// TIA Portal V15.1 export
// export: Created 2024-06-21T08:41:23.5653437Z, ExportSetting WithDefaults, DisplayName Totally Integrated Automation Portal, DisplayVersion V15.1 Update 5, DisplayName TIA Portal Openness, DisplayVersion V15.1 Update 5, DisplayName SINAMICS Startdrive Advanced, DisplayVersion V15.1, DisplayName G130, G150, S120, S150, SINAMICS MV, S210, DisplayVersion V15.1, DisplayName G110M, G120, G120C, G120D, G120P, DisplayVersion V15.1, DisplayName STEP 7 Professional, DisplayVersion V15.1 Update 5, DisplayName STEP 7 Safety, DisplayVersion V15.1, DisplayName WinCC Professional, DisplayVersion V15.1 Update 5, DisplayName SIMATIC Visualization Architect, DisplayVersion V15.1
FUNCTION "209210ZS01AS" : Void   // FC322, FBD
TITLE = 209210ZS01AS Panels
{ S7_Optimized_Access := 'TRUE' }
AUTHOR : VCC
VERSION : 0.1
// stored: AutoNumber false, IsIECCheckEnabled false, SetENOAutomatically False, UDAEnableTagReadback false
   VAR_OUTPUT
      O_AlarmA : Bool;   // Alarm A
      O_AlarmB : Bool;   // Alarm B
      O_AlarmC : Bool;   // Alarm C
      O_AlarmD : Bool;   // Alarm D
      O_AlarmABCondition : Bool;   // Alarm AB condition
      H_IAnim : Word;   // For animation of icon
   END_VAR
BEGIN

REGION Network 1: **** --------------------- Pushbuttons Equipment 209210AS10 --------------------- ****
END_REGION

REGION Network 2: **** 4.3 - Machine status - Operator Selection **** Pushbutton 210CHB21 Holdback Down
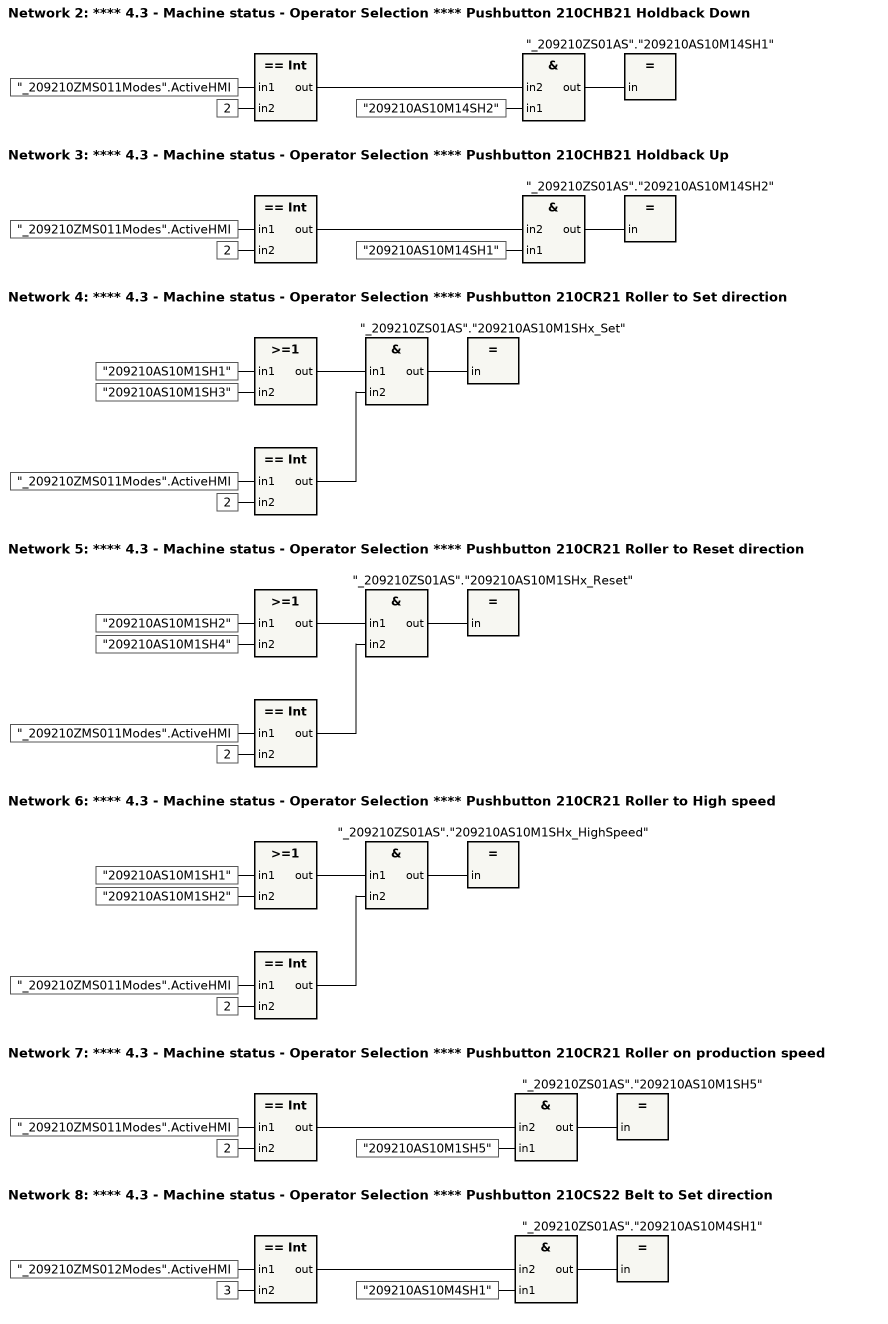
   "_209210ZS01AS"."209210AS10M14SH1" := ("_209210ZMS011Modes".ActiveHMI = 2) AND "209210AS10M14SH2";
END_REGION

REGION Network 3: **** 4.3 - Machine status - Operator Selection **** Pushbutton 210CHB21 Holdback Up
   "_209210ZS01AS"."209210AS10M14SH2" := ("_209210ZMS011Modes".ActiveHMI = 2) AND "209210AS10M14SH1";
END_REGION

REGION Network 4: **** 4.3 - Machine status - Operator Selection **** Pushbutton 210CR21 Roller to Set direction
   "_209210ZS01AS"."209210AS10M1SHx_Set" := ("209210AS10M1SH1" OR "209210AS10M1SH3") AND ("_209210ZMS011Modes".ActiveHMI = 2);
END_REGION

REGION Network 5: **** 4.3 - Machine status - Operator Selection **** Pushbutton 210CR21 Roller to Reset direction
   "_209210ZS01AS"."209210AS10M1SHx_Reset" := ("209210AS10M1SH2" OR "209210AS10M1SH4") AND ("_209210ZMS011Modes".ActiveHMI = 2);
END_REGION

REGION Network 6: **** 4.3 - Machine status - Operator Selection **** Pushbutton 210CR21 Roller to High speed
   "_209210ZS01AS"."209210AS10M1SHx_HighSpeed" := ("209210AS10M1SH1" OR "209210AS10M1SH2") AND ("_209210ZMS011Modes".ActiveHMI = 2);
END_REGION

REGION Network 7: **** 4.3 - Machine status - Operator Selection **** Pushbutton 210CR21 Roller on production speed
   "_209210ZS01AS"."209210AS10M1SH5" := ("_209210ZMS011Modes".ActiveHMI = 2) AND "209210AS10M1SH5";
END_REGION

REGION Network 8: **** 4.3 - Machine status - Operator Selection **** Pushbutton 210CS22 Belt to Set direction
   "_209210ZS01AS"."209210AS10M4SH1" := ("_209210ZMS012Modes".ActiveHMI = 3) AND "209210AS10M4SH1";
END_REGION

REGION Network 9: **** 4.3 - Machine status - Operator Selection **** Pushbutton 210CS22 Belt to Reset direction
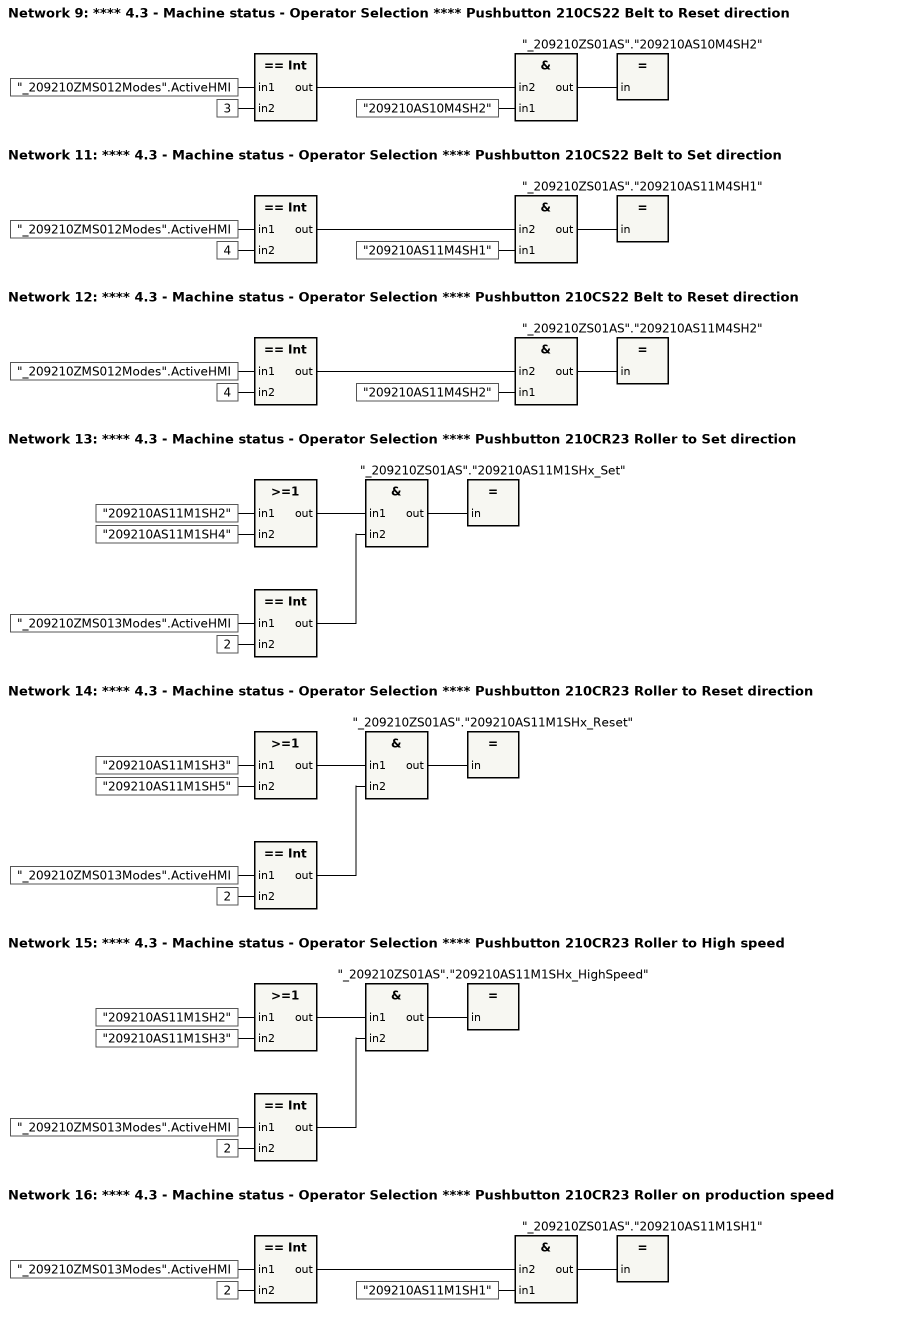
   "_209210ZS01AS"."209210AS10M4SH2" := ("_209210ZMS012Modes".ActiveHMI = 3) AND "209210AS10M4SH2";
END_REGION

REGION Network 10: **** --------------------- Pushbuttons Equipment 209210AS11 --------------------- ****
END_REGION

REGION Network 11: **** 4.3 - Machine status - Operator Selection **** Pushbutton 210CS22 Belt to Set direction
   "_209210ZS01AS"."209210AS11M4SH1" := ("_209210ZMS012Modes".ActiveHMI = 4) AND "209210AS11M4SH1";
END_REGION

REGION Network 12: **** 4.3 - Machine status - Operator Selection **** Pushbutton 210CS22 Belt to Reset direction
   "_209210ZS01AS"."209210AS11M4SH2" := ("_209210ZMS012Modes".ActiveHMI = 4) AND "209210AS11M4SH2";
END_REGION

REGION Network 13: **** 4.3 - Machine status - Operator Selection **** Pushbutton 210CR23 Roller to Set direction
   "_209210ZS01AS"."209210AS11M1SHx_Set" := ("209210AS11M1SH2" OR "209210AS11M1SH4") AND ("_209210ZMS013Modes".ActiveHMI = 2);
END_REGION

REGION Network 14: **** 4.3 - Machine status - Operator Selection **** Pushbutton 210CR23 Roller to Reset direction
   "_209210ZS01AS"."209210AS11M1SHx_Reset" := ("209210AS11M1SH3" OR "209210AS11M1SH5") AND ("_209210ZMS013Modes".ActiveHMI = 2);
END_REGION

REGION Network 15: **** 4.3 - Machine status - Operator Selection **** Pushbutton 210CR23 Roller to High speed
   "_209210ZS01AS"."209210AS11M1SHx_HighSpeed" := ("209210AS11M1SH2" OR "209210AS11M1SH3") AND ("_209210ZMS013Modes".ActiveHMI = 2);
END_REGION

REGION Network 16: **** 4.3 - Machine status - Operator Selection **** Pushbutton 210CR23 Roller on production speed
   "_209210ZS01AS"."209210AS11M1SH1" := ("_209210ZMS013Modes".ActiveHMI = 2) AND "209210AS11M1SH1";
END_REGION

REGION Network 17: **** -------------------------------------------------- ****
END_REGION

REGION Network 18: **** 4.6 - Machine status - Indications **** Icon animation
   // Icon animation
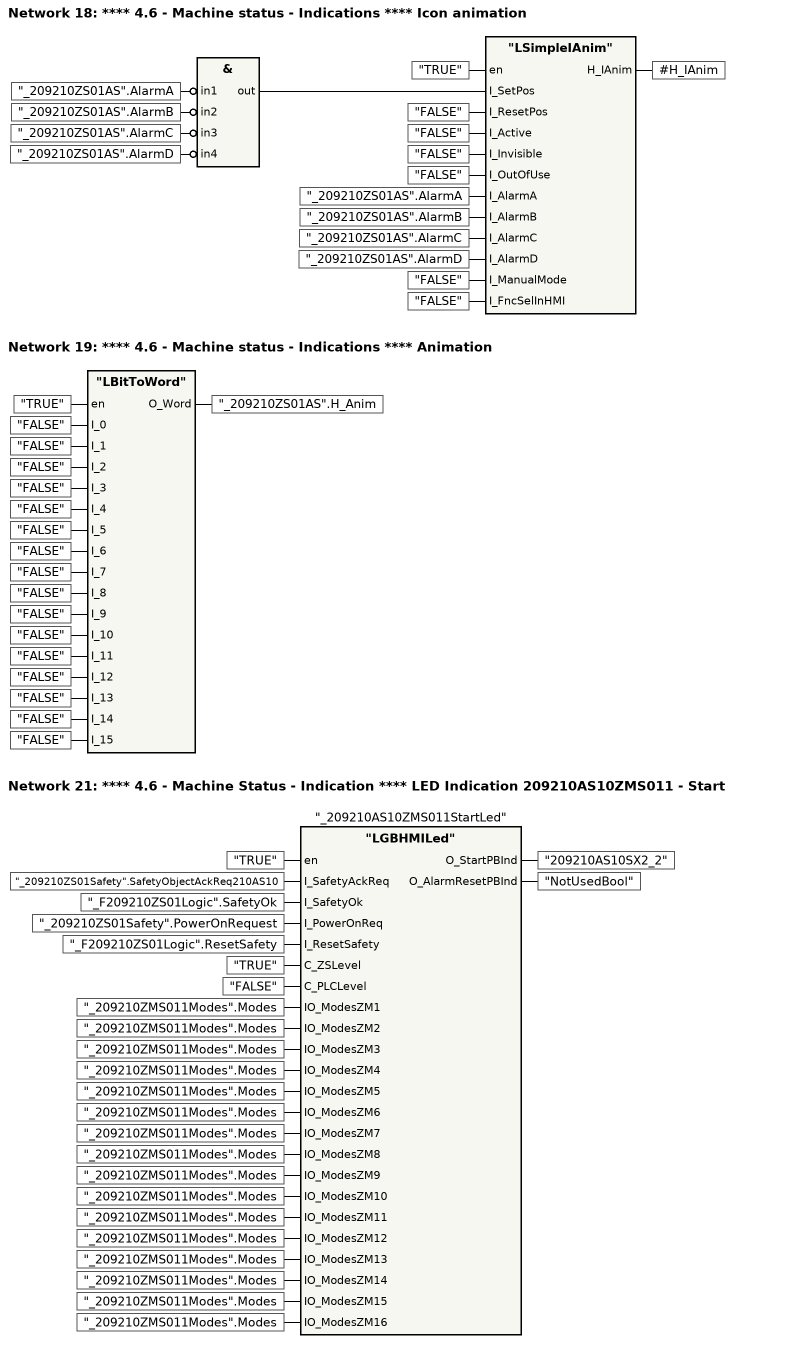
   IF "TRUE" THEN
       "LSimpleIAnim"(I_SetPos := NOT "_209210ZS01AS".AlarmA AND NOT "_209210ZS01AS".AlarmB AND NOT "_209210ZS01AS".AlarmC AND NOT "_209210ZS01AS".AlarmD,
                      I_ResetPos := "FALSE",
                      I_Active := "FALSE",
                      I_Invisible := "FALSE",
                      I_OutOfUse := "FALSE",
                      I_AlarmA := "_209210ZS01AS".AlarmA,
                      I_AlarmB := "_209210ZS01AS".AlarmB,
                      I_AlarmC := "_209210ZS01AS".AlarmC,
                      I_AlarmD := "_209210ZS01AS".AlarmD,
                      I_ManualMode := "FALSE",
                      I_FncSelInHMI := "FALSE",
                      H_IAnim => #H_IAnim);
   END_IF;
END_REGION

REGION Network 19: **** 4.6 - Machine status - Indications **** Animation
   // Animation
   IF "TRUE" THEN
       "LBitToWord"(I_0 := "FALSE",
                    I_1 := "FALSE",
                    I_2 := "FALSE",
                    I_3 := "FALSE",
                    I_4 := "FALSE",
                    I_5 := "FALSE",
                    I_6 := "FALSE",
                    I_7 := "FALSE",
                    I_8 := "FALSE",
                    I_9 := "FALSE",
                    I_10 := "FALSE",
                    I_11 := "FALSE",
                    I_12 := "FALSE",
                    I_13 := "FALSE",
                    I_14 := "FALSE",
                    I_15 := "FALSE",
                    O_Word => "_209210ZS01AS".H_Anim);
   END_IF;
END_REGION

NETWORK
TITLE = **** 4.6 - Machine Status - Indications **** Animation DB number
// DB number
      OPN   "_209210ZS01AS";
      L     DBNO;
      T     "_209210ZS01AS".H_DBnr;

REGION Network 21: **** 4.6 - Machine Status - Indication **** LED Indication 209210AS10ZMS011 - Start
   // The Module handles indications for Start and Reset buttons
   IF "TRUE" THEN
       "_209210AS10ZMS011StartLed"(I_SafetyAckReq := "_209210ZS01Safety".SafetyObjectAckReq210AS10,   // "LGBHMILed"
                               I_SafetyOk := "_F209210ZS01Logic".SafetyOk,
                               I_PowerOnReq := "_209210ZS01Safety".PowerOnRequest,
                               I_ResetSafety := "_F209210ZS01Logic".ResetSafety,
                               C_ZSLevel := "TRUE",
                               C_PLCLevel := "FALSE",
                               IO_ModesZM1 := "_209210ZMS011Modes".Modes,
                               IO_ModesZM2 := "_209210ZMS011Modes".Modes,
                               IO_ModesZM3 := "_209210ZMS011Modes".Modes,
                               IO_ModesZM4 := "_209210ZMS011Modes".Modes,
                               IO_ModesZM5 := "_209210ZMS011Modes".Modes,
                               IO_ModesZM6 := "_209210ZMS011Modes".Modes,
                               IO_ModesZM7 := "_209210ZMS011Modes".Modes,
                               IO_ModesZM8 := "_209210ZMS011Modes".Modes,
                               IO_ModesZM9 := "_209210ZMS011Modes".Modes,
                               IO_ModesZM10 := "_209210ZMS011Modes".Modes,
                               IO_ModesZM11 := "_209210ZMS011Modes".Modes,
                               IO_ModesZM12 := "_209210ZMS011Modes".Modes,
                               IO_ModesZM13 := "_209210ZMS011Modes".Modes,
                               IO_ModesZM14 := "_209210ZMS011Modes".Modes,
                               IO_ModesZM15 := "_209210ZMS011Modes".Modes,
                               IO_ModesZM16 := "_209210ZMS011Modes".Modes,
                               O_StartPBInd => "209210AS10SX2_2",
                               O_AlarmResetPBInd => "NotUsedBool");
   END_IF;
END_REGION

REGION Network 22: **** 4.6 - Machine Status - Indication **** LED Indication 209210AS10ZMS012 - Start
   // The Module handles indications for Start and Reset buttons
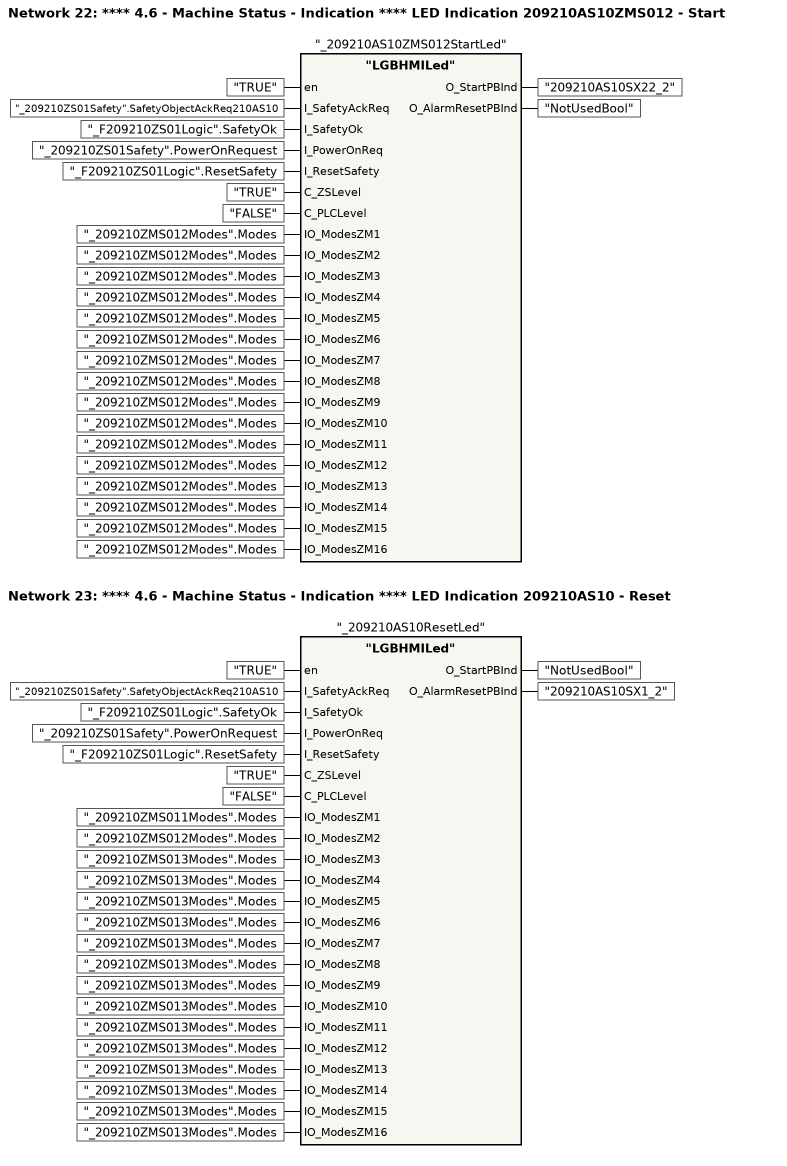
   IF "TRUE" THEN
       "_209210AS10ZMS012StartLed"(I_SafetyAckReq := "_209210ZS01Safety".SafetyObjectAckReq210AS10,   // "LGBHMILed"
                               I_SafetyOk := "_F209210ZS01Logic".SafetyOk,
                               I_PowerOnReq := "_209210ZS01Safety".PowerOnRequest,
                               I_ResetSafety := "_F209210ZS01Logic".ResetSafety,
                               C_ZSLevel := "TRUE",
                               C_PLCLevel := "FALSE",
                               IO_ModesZM1 := "_209210ZMS012Modes".Modes,
                               IO_ModesZM2 := "_209210ZMS012Modes".Modes,
                               IO_ModesZM3 := "_209210ZMS012Modes".Modes,
                               IO_ModesZM4 := "_209210ZMS012Modes".Modes,
                               IO_ModesZM5 := "_209210ZMS012Modes".Modes,
                               IO_ModesZM6 := "_209210ZMS012Modes".Modes,
                               IO_ModesZM7 := "_209210ZMS012Modes".Modes,
                               IO_ModesZM8 := "_209210ZMS012Modes".Modes,
                               IO_ModesZM9 := "_209210ZMS012Modes".Modes,
                               IO_ModesZM10 := "_209210ZMS012Modes".Modes,
                               IO_ModesZM11 := "_209210ZMS012Modes".Modes,
                               IO_ModesZM12 := "_209210ZMS012Modes".Modes,
                               IO_ModesZM13 := "_209210ZMS012Modes".Modes,
                               IO_ModesZM14 := "_209210ZMS012Modes".Modes,
                               IO_ModesZM15 := "_209210ZMS012Modes".Modes,
                               IO_ModesZM16 := "_209210ZMS012Modes".Modes,
                               O_StartPBInd => "209210AS10SX22_2",
                               O_AlarmResetPBInd => "NotUsedBool");
   END_IF;
END_REGION

REGION Network 23: **** 4.6 - Machine Status - Indication **** LED Indication 209210AS10 - Reset
   // The Module handles indications for Start and Reset buttons
   IF "TRUE" THEN
       "_209210AS10ResetLed"(I_SafetyAckReq := "_209210ZS01Safety".SafetyObjectAckReq210AS10,   // "LGBHMILed"
                             I_SafetyOk := "_F209210ZS01Logic".SafetyOk,
                             I_PowerOnReq := "_209210ZS01Safety".PowerOnRequest,
                             I_ResetSafety := "_F209210ZS01Logic".ResetSafety,
                             C_ZSLevel := "TRUE",
                             C_PLCLevel := "FALSE",
                             IO_ModesZM1 := "_209210ZMS011Modes".Modes,
                             IO_ModesZM2 := "_209210ZMS012Modes".Modes,
                             IO_ModesZM3 := "_209210ZMS013Modes".Modes,
                             IO_ModesZM4 := "_209210ZMS013Modes".Modes,
                             IO_ModesZM5 := "_209210ZMS013Modes".Modes,
                             IO_ModesZM6 := "_209210ZMS013Modes".Modes,
                             IO_ModesZM7 := "_209210ZMS013Modes".Modes,
                             IO_ModesZM8 := "_209210ZMS013Modes".Modes,
                             IO_ModesZM9 := "_209210ZMS013Modes".Modes,
                             IO_ModesZM10 := "_209210ZMS013Modes".Modes,
                             IO_ModesZM11 := "_209210ZMS013Modes".Modes,
                             IO_ModesZM12 := "_209210ZMS013Modes".Modes,
                             IO_ModesZM13 := "_209210ZMS013Modes".Modes,
                             IO_ModesZM14 := "_209210ZMS013Modes".Modes,
                             IO_ModesZM15 := "_209210ZMS013Modes".Modes,
                             IO_ModesZM16 := "_209210ZMS013Modes".Modes,
                             O_StartPBInd => "NotUsedBool",
                             O_AlarmResetPBInd => "209210AS10SX1_2");
   END_IF;
END_REGION

REGION Network 24: **** 4.6 - Machine Status - Indication **** LED Indication 209210AS11ZMS012 - Start
   // The Module handles indications for Start and Reset buttons
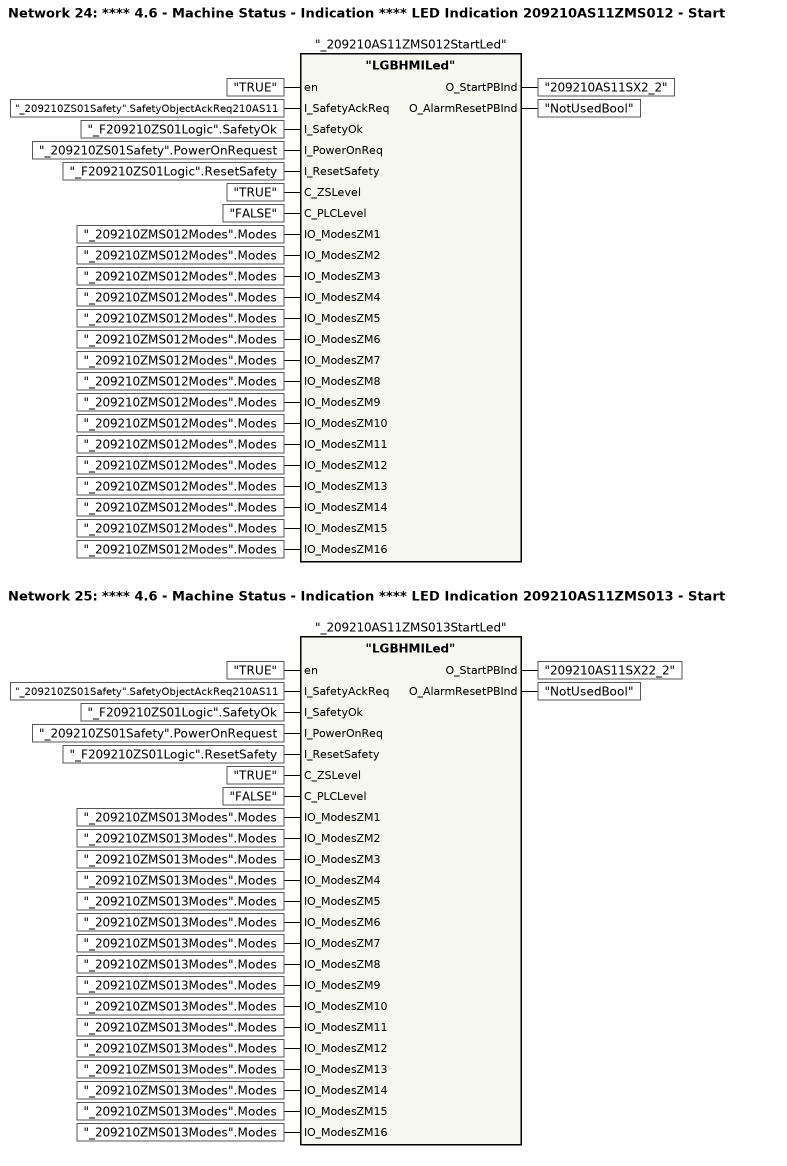
   IF "TRUE" THEN
       "_209210AS11ZMS012StartLed"(I_SafetyAckReq := "_209210ZS01Safety".SafetyObjectAckReq210AS11,   // "LGBHMILed"
                               I_SafetyOk := "_F209210ZS01Logic".SafetyOk,
                               I_PowerOnReq := "_209210ZS01Safety".PowerOnRequest,
                               I_ResetSafety := "_F209210ZS01Logic".ResetSafety,
                               C_ZSLevel := "TRUE",
                               C_PLCLevel := "FALSE",
                               IO_ModesZM1 := "_209210ZMS012Modes".Modes,
                               IO_ModesZM2 := "_209210ZMS012Modes".Modes,
                               IO_ModesZM3 := "_209210ZMS012Modes".Modes,
                               IO_ModesZM4 := "_209210ZMS012Modes".Modes,
                               IO_ModesZM5 := "_209210ZMS012Modes".Modes,
                               IO_ModesZM6 := "_209210ZMS012Modes".Modes,
                               IO_ModesZM7 := "_209210ZMS012Modes".Modes,
                               IO_ModesZM8 := "_209210ZMS012Modes".Modes,
                               IO_ModesZM9 := "_209210ZMS012Modes".Modes,
                               IO_ModesZM10 := "_209210ZMS012Modes".Modes,
                               IO_ModesZM11 := "_209210ZMS012Modes".Modes,
                               IO_ModesZM12 := "_209210ZMS012Modes".Modes,
                               IO_ModesZM13 := "_209210ZMS012Modes".Modes,
                               IO_ModesZM14 := "_209210ZMS012Modes".Modes,
                               IO_ModesZM15 := "_209210ZMS012Modes".Modes,
                               IO_ModesZM16 := "_209210ZMS012Modes".Modes,
                               O_StartPBInd => "209210AS11SX2_2",
                               O_AlarmResetPBInd => "NotUsedBool");
   END_IF;
END_REGION

REGION Network 25: **** 4.6 - Machine Status - Indication **** LED Indication 209210AS11ZMS013 - Start
   // The Module handles indications for Start and Reset buttons
   IF "TRUE" THEN
       "_209210AS11ZMS013StartLed"(I_SafetyAckReq := "_209210ZS01Safety".SafetyObjectAckReq210AS11,   // "LGBHMILed"
                               I_SafetyOk := "_F209210ZS01Logic".SafetyOk,
                               I_PowerOnReq := "_209210ZS01Safety".PowerOnRequest,
                               I_ResetSafety := "_F209210ZS01Logic".ResetSafety,
                               C_ZSLevel := "TRUE",
                               C_PLCLevel := "FALSE",
                               IO_ModesZM1 := "_209210ZMS013Modes".Modes,
                               IO_ModesZM2 := "_209210ZMS013Modes".Modes,
                               IO_ModesZM3 := "_209210ZMS013Modes".Modes,
                               IO_ModesZM4 := "_209210ZMS013Modes".Modes,
                               IO_ModesZM5 := "_209210ZMS013Modes".Modes,
                               IO_ModesZM6 := "_209210ZMS013Modes".Modes,
                               IO_ModesZM7 := "_209210ZMS013Modes".Modes,
                               IO_ModesZM8 := "_209210ZMS013Modes".Modes,
                               IO_ModesZM9 := "_209210ZMS013Modes".Modes,
                               IO_ModesZM10 := "_209210ZMS013Modes".Modes,
                               IO_ModesZM11 := "_209210ZMS013Modes".Modes,
                               IO_ModesZM12 := "_209210ZMS013Modes".Modes,
                               IO_ModesZM13 := "_209210ZMS013Modes".Modes,
                               IO_ModesZM14 := "_209210ZMS013Modes".Modes,
                               IO_ModesZM15 := "_209210ZMS013Modes".Modes,
                               IO_ModesZM16 := "_209210ZMS013Modes".Modes,
                               O_StartPBInd => "209210AS11SX22_2",
                               O_AlarmResetPBInd => "NotUsedBool");
   END_IF;
END_REGION

REGION Network 26: **** 4.6 - Machine Status - Indication **** LED Indication 209210AS11 - Reset
   // The Module handles indications for Start and Reset buttons
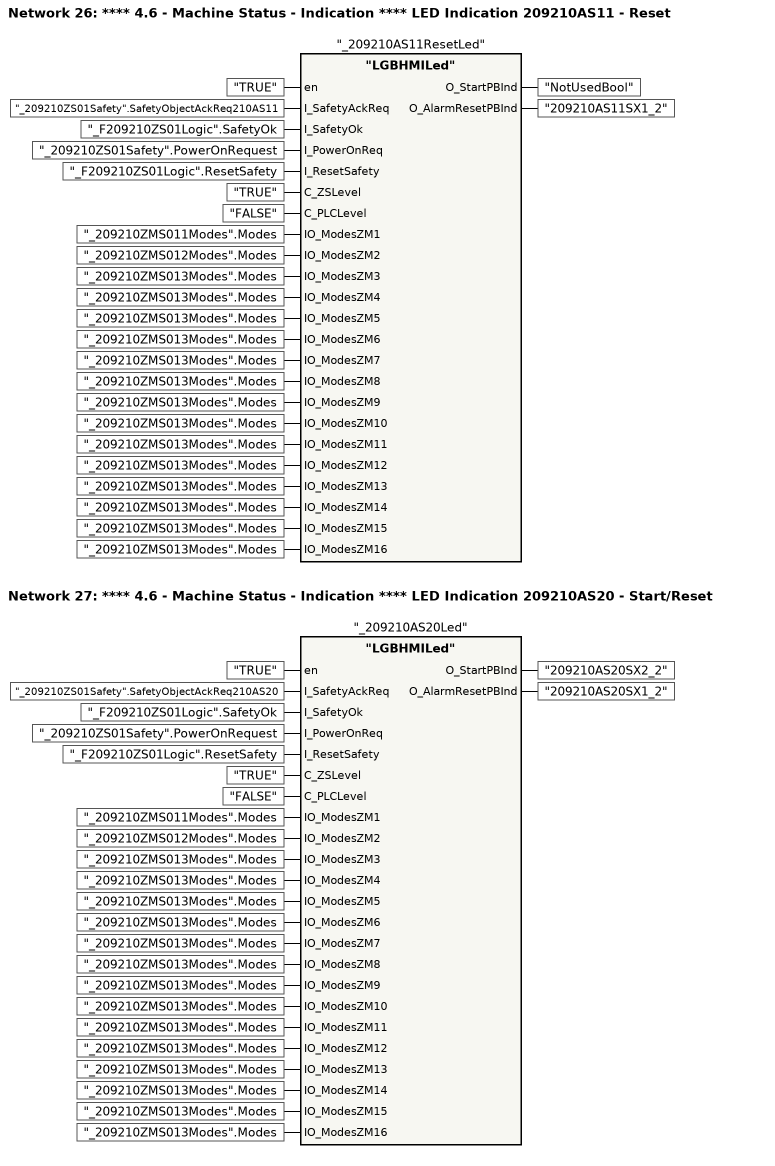
   IF "TRUE" THEN
       "_209210AS11ResetLed"(I_SafetyAckReq := "_209210ZS01Safety".SafetyObjectAckReq210AS11,   // "LGBHMILed"
                             I_SafetyOk := "_F209210ZS01Logic".SafetyOk,
                             I_PowerOnReq := "_209210ZS01Safety".PowerOnRequest,
                             I_ResetSafety := "_F209210ZS01Logic".ResetSafety,
                             C_ZSLevel := "TRUE",
                             C_PLCLevel := "FALSE",
                             IO_ModesZM1 := "_209210ZMS011Modes".Modes,
                             IO_ModesZM2 := "_209210ZMS012Modes".Modes,
                             IO_ModesZM3 := "_209210ZMS013Modes".Modes,
                             IO_ModesZM4 := "_209210ZMS013Modes".Modes,
                             IO_ModesZM5 := "_209210ZMS013Modes".Modes,
                             IO_ModesZM6 := "_209210ZMS013Modes".Modes,
                             IO_ModesZM7 := "_209210ZMS013Modes".Modes,
                             IO_ModesZM8 := "_209210ZMS013Modes".Modes,
                             IO_ModesZM9 := "_209210ZMS013Modes".Modes,
                             IO_ModesZM10 := "_209210ZMS013Modes".Modes,
                             IO_ModesZM11 := "_209210ZMS013Modes".Modes,
                             IO_ModesZM12 := "_209210ZMS013Modes".Modes,
                             IO_ModesZM13 := "_209210ZMS013Modes".Modes,
                             IO_ModesZM14 := "_209210ZMS013Modes".Modes,
                             IO_ModesZM15 := "_209210ZMS013Modes".Modes,
                             IO_ModesZM16 := "_209210ZMS013Modes".Modes,
                             O_StartPBInd => "NotUsedBool",
                             O_AlarmResetPBInd => "209210AS11SX1_2");
   END_IF;
END_REGION

REGION Network 27: **** 4.6 - Machine Status - Indication **** LED Indication 209210AS20 - Start/Reset
   // The Module handles indications for Start and Reset buttons
   IF "TRUE" THEN
       "_209210AS20Led"(I_SafetyAckReq := "_209210ZS01Safety".SafetyObjectAckReq210AS20,   // "LGBHMILed"
                        I_SafetyOk := "_F209210ZS01Logic".SafetyOk,
                        I_PowerOnReq := "_209210ZS01Safety".PowerOnRequest,
                        I_ResetSafety := "_F209210ZS01Logic".ResetSafety,
                        C_ZSLevel := "TRUE",
                        C_PLCLevel := "FALSE",
                        IO_ModesZM1 := "_209210ZMS011Modes".Modes,
                        IO_ModesZM2 := "_209210ZMS012Modes".Modes,
                        IO_ModesZM3 := "_209210ZMS013Modes".Modes,
                        IO_ModesZM4 := "_209210ZMS013Modes".Modes,
                        IO_ModesZM5 := "_209210ZMS013Modes".Modes,
                        IO_ModesZM6 := "_209210ZMS013Modes".Modes,
                        IO_ModesZM7 := "_209210ZMS013Modes".Modes,
                        IO_ModesZM8 := "_209210ZMS013Modes".Modes,
                        IO_ModesZM9 := "_209210ZMS013Modes".Modes,
                        IO_ModesZM10 := "_209210ZMS013Modes".Modes,
                        IO_ModesZM11 := "_209210ZMS013Modes".Modes,
                        IO_ModesZM12 := "_209210ZMS013Modes".Modes,
                        IO_ModesZM13 := "_209210ZMS013Modes".Modes,
                        IO_ModesZM14 := "_209210ZMS013Modes".Modes,
                        IO_ModesZM15 := "_209210ZMS013Modes".Modes,
                        IO_ModesZM16 := "_209210ZMS013Modes".Modes,
                        O_StartPBInd => "209210AS20SX2_2",
                        O_AlarmResetPBInd => "209210AS20SX1_2");
   END_IF;
END_REGION

REGION Network 28: **** 4.6 - Machine Status - Indication **** LED Indication 209210AS40 - Start/Reset
   // The Module handles indications for Start and Reset buttons
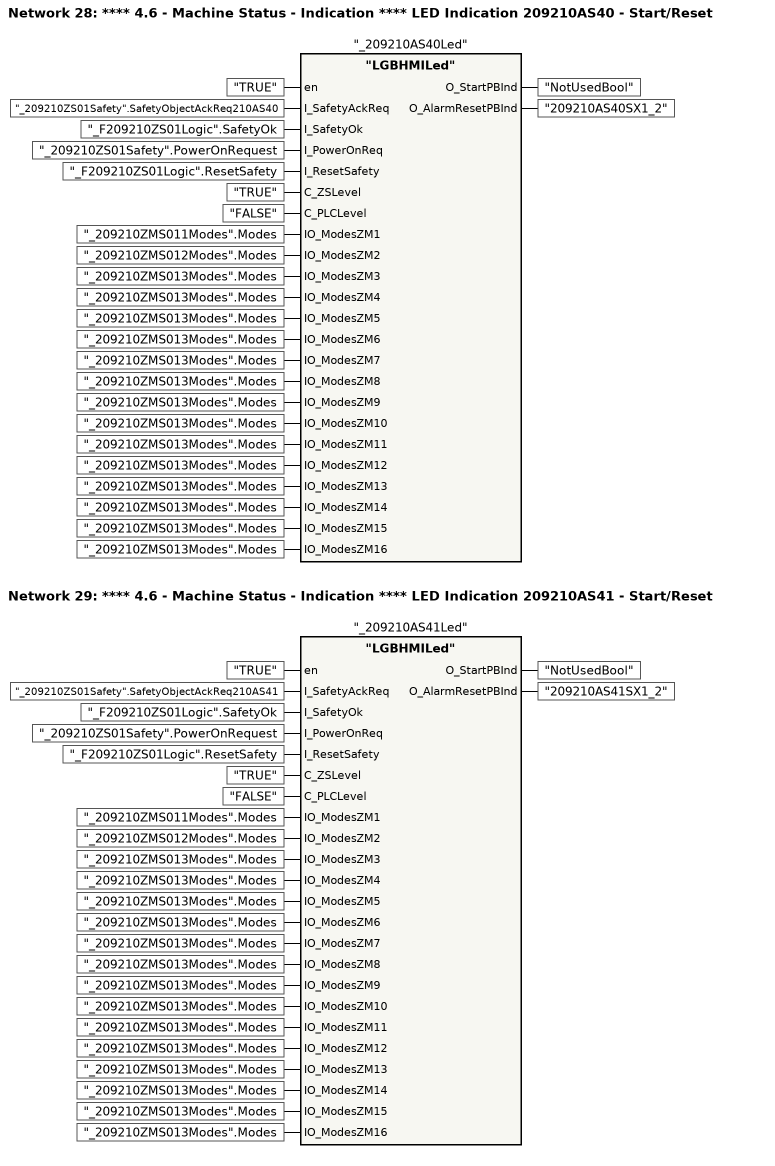
   IF "TRUE" THEN
       "_209210AS40Led"(I_SafetyAckReq := "_209210ZS01Safety".SafetyObjectAckReq210AS40,   // "LGBHMILed"
                        I_SafetyOk := "_F209210ZS01Logic".SafetyOk,
                        I_PowerOnReq := "_209210ZS01Safety".PowerOnRequest,
                        I_ResetSafety := "_F209210ZS01Logic".ResetSafety,
                        C_ZSLevel := "TRUE",
                        C_PLCLevel := "FALSE",
                        IO_ModesZM1 := "_209210ZMS011Modes".Modes,
                        IO_ModesZM2 := "_209210ZMS012Modes".Modes,
                        IO_ModesZM3 := "_209210ZMS013Modes".Modes,
                        IO_ModesZM4 := "_209210ZMS013Modes".Modes,
                        IO_ModesZM5 := "_209210ZMS013Modes".Modes,
                        IO_ModesZM6 := "_209210ZMS013Modes".Modes,
                        IO_ModesZM7 := "_209210ZMS013Modes".Modes,
                        IO_ModesZM8 := "_209210ZMS013Modes".Modes,
                        IO_ModesZM9 := "_209210ZMS013Modes".Modes,
                        IO_ModesZM10 := "_209210ZMS013Modes".Modes,
                        IO_ModesZM11 := "_209210ZMS013Modes".Modes,
                        IO_ModesZM12 := "_209210ZMS013Modes".Modes,
                        IO_ModesZM13 := "_209210ZMS013Modes".Modes,
                        IO_ModesZM14 := "_209210ZMS013Modes".Modes,
                        IO_ModesZM15 := "_209210ZMS013Modes".Modes,
                        IO_ModesZM16 := "_209210ZMS013Modes".Modes,
                        O_StartPBInd => "NotUsedBool",
                        O_AlarmResetPBInd => "209210AS40SX1_2");
   END_IF;
END_REGION

REGION Network 29: **** 4.6 - Machine Status - Indication **** LED Indication 209210AS41 - Start/Reset
   // The Module handles indications for Start and Reset buttons
   IF "TRUE" THEN
       "_209210AS41Led"(I_SafetyAckReq := "_209210ZS01Safety".SafetyObjectAckReq210AS41,   // "LGBHMILed"
                        I_SafetyOk := "_F209210ZS01Logic".SafetyOk,
                        I_PowerOnReq := "_209210ZS01Safety".PowerOnRequest,
                        I_ResetSafety := "_F209210ZS01Logic".ResetSafety,
                        C_ZSLevel := "TRUE",
                        C_PLCLevel := "FALSE",
                        IO_ModesZM1 := "_209210ZMS011Modes".Modes,
                        IO_ModesZM2 := "_209210ZMS012Modes".Modes,
                        IO_ModesZM3 := "_209210ZMS013Modes".Modes,
                        IO_ModesZM4 := "_209210ZMS013Modes".Modes,
                        IO_ModesZM5 := "_209210ZMS013Modes".Modes,
                        IO_ModesZM6 := "_209210ZMS013Modes".Modes,
                        IO_ModesZM7 := "_209210ZMS013Modes".Modes,
                        IO_ModesZM8 := "_209210ZMS013Modes".Modes,
                        IO_ModesZM9 := "_209210ZMS013Modes".Modes,
                        IO_ModesZM10 := "_209210ZMS013Modes".Modes,
                        IO_ModesZM11 := "_209210ZMS013Modes".Modes,
                        IO_ModesZM12 := "_209210ZMS013Modes".Modes,
                        IO_ModesZM13 := "_209210ZMS013Modes".Modes,
                        IO_ModesZM14 := "_209210ZMS013Modes".Modes,
                        IO_ModesZM15 := "_209210ZMS013Modes".Modes,
                        IO_ModesZM16 := "_209210ZMS013Modes".Modes,
                        O_StartPBInd => "NotUsedBool",
                        O_AlarmResetPBInd => "209210AS41SX1_2");
   END_IF;
END_REGION

REGION Network 30: **** 4.6 - Machine Status - Indication **** LED Indication 209210ASH01 - Start/Reset
   // The Module handles indications for Start and Reset buttons
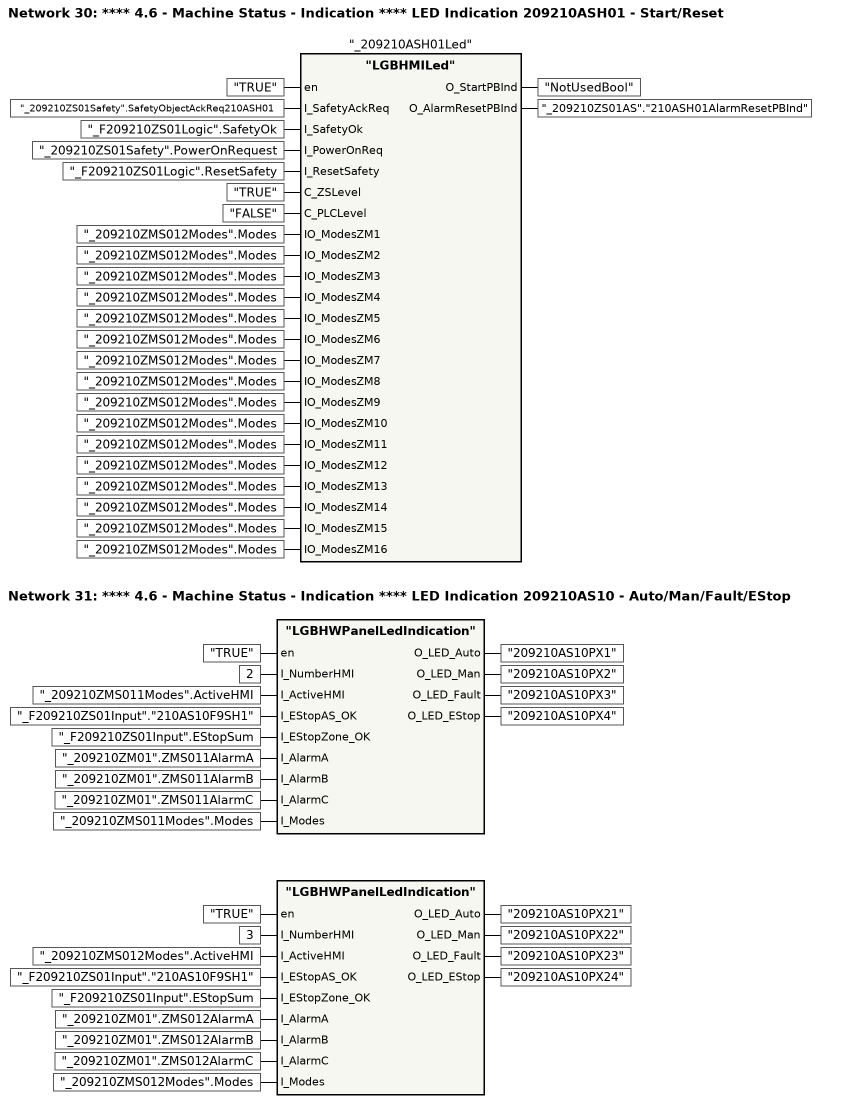
   IF "TRUE" THEN
       "_209210ASH01Led"(I_SafetyAckReq := "_209210ZS01Safety".SafetyObjectAckReq210ASH01,   // "LGBHMILed"
                         I_SafetyOk := "_F209210ZS01Logic".SafetyOk,
                         I_PowerOnReq := "_209210ZS01Safety".PowerOnRequest,
                         I_ResetSafety := "_F209210ZS01Logic".ResetSafety,
                         C_ZSLevel := "TRUE",
                         C_PLCLevel := "FALSE",
                         IO_ModesZM1 := "_209210ZMS012Modes".Modes,
                         IO_ModesZM2 := "_209210ZMS012Modes".Modes,
                         IO_ModesZM3 := "_209210ZMS012Modes".Modes,
                         IO_ModesZM4 := "_209210ZMS012Modes".Modes,
                         IO_ModesZM5 := "_209210ZMS012Modes".Modes,
                         IO_ModesZM6 := "_209210ZMS012Modes".Modes,
                         IO_ModesZM7 := "_209210ZMS012Modes".Modes,
                         IO_ModesZM8 := "_209210ZMS012Modes".Modes,
                         IO_ModesZM9 := "_209210ZMS012Modes".Modes,
                         IO_ModesZM10 := "_209210ZMS012Modes".Modes,
                         IO_ModesZM11 := "_209210ZMS012Modes".Modes,
                         IO_ModesZM12 := "_209210ZMS012Modes".Modes,
                         IO_ModesZM13 := "_209210ZMS012Modes".Modes,
                         IO_ModesZM14 := "_209210ZMS012Modes".Modes,
                         IO_ModesZM15 := "_209210ZMS012Modes".Modes,
                         IO_ModesZM16 := "_209210ZMS012Modes".Modes,
                         O_StartPBInd => "NotUsedBool",
                         O_AlarmResetPBInd => "_209210ZS01AS"."210ASH01AlarmResetPBInd");
   END_IF;
END_REGION

REGION Network 31: **** 4.6 - Machine Status - Indication **** LED Indication 209210AS10 - Auto/Man/Fault/EStop
   IF "TRUE" THEN
       "LGBHWPanelLedIndication"(I_NumberHMI := 2,
                               I_ActiveHMI := "_209210ZMS011Modes".ActiveHMI,
                               I_EStopAS_OK := "_F209210ZS01Input"."210AS10F9SH1",
                               I_EStopZone_OK := "_F209210ZS01Input".EStopSum,
                               I_AlarmA := "_209210ZM01".ZMS011AlarmA,
                               I_AlarmB := "_209210ZM01".ZMS011AlarmB,
                               I_AlarmC := "_209210ZM01".ZMS011AlarmC,
                               I_Modes := "_209210ZMS011Modes".Modes,
                               O_LED_Auto => "209210AS10PX1",
                               O_LED_Man => "209210AS10PX2",
                               O_LED_Fault => "209210AS10PX3",
                               O_LED_EStop => "209210AS10PX4");
   END_IF;
   IF "TRUE" THEN
       "LGBHWPanelLedIndication"(I_NumberHMI := 3,
                               I_ActiveHMI := "_209210ZMS012Modes".ActiveHMI,
                               I_EStopAS_OK := "_F209210ZS01Input"."210AS10F9SH1",
                               I_EStopZone_OK := "_F209210ZS01Input".EStopSum,
                               I_AlarmA := "_209210ZM01".ZMS012AlarmA,
                               I_AlarmB := "_209210ZM01".ZMS012AlarmB,
                               I_AlarmC := "_209210ZM01".ZMS012AlarmC,
                               I_Modes := "_209210ZMS012Modes".Modes,
                               O_LED_Auto => "209210AS10PX21",
                               O_LED_Man => "209210AS10PX22",
                               O_LED_Fault => "209210AS10PX23",
                               O_LED_EStop => "209210AS10PX24");
   END_IF;
END_REGION

REGION Network 32: **** 4.6 - Machine Status - Indication **** LED Indication 209210AS11 - Auto/Man/Fault/EStop
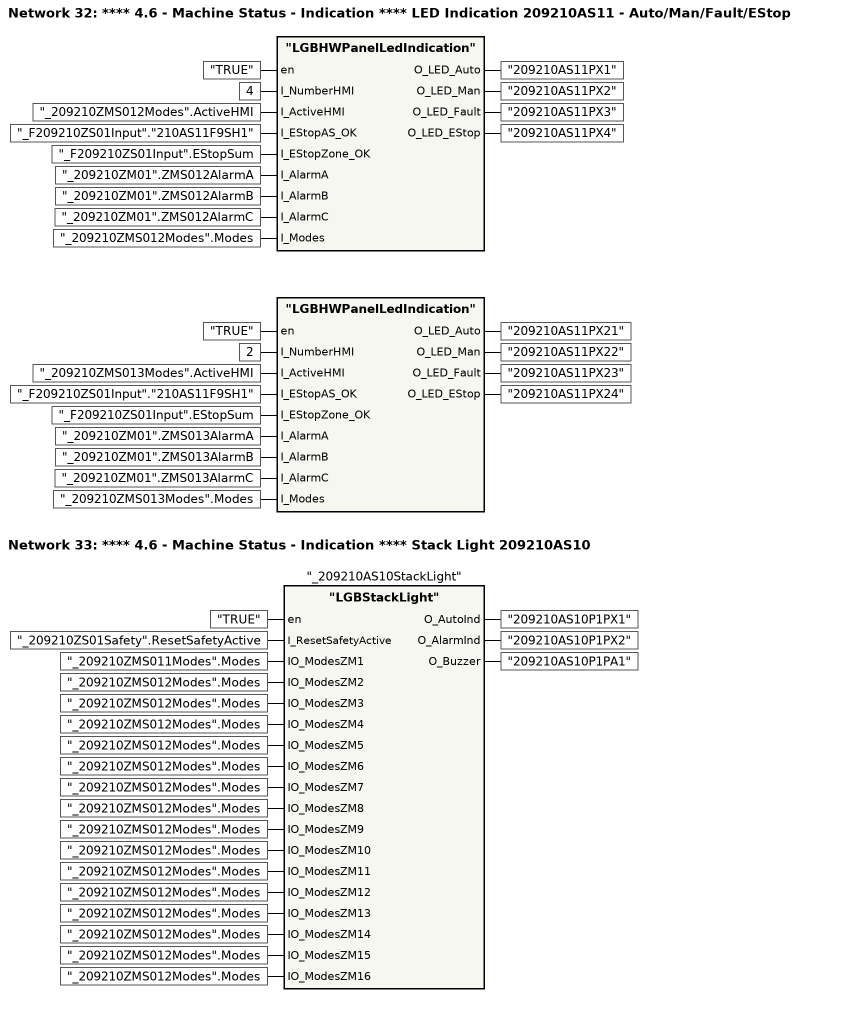
   IF "TRUE" THEN
       "LGBHWPanelLedIndication"(I_NumberHMI := 4,
                               I_ActiveHMI := "_209210ZMS012Modes".ActiveHMI,
                               I_EStopAS_OK := "_F209210ZS01Input"."210AS11F9SH1",
                               I_EStopZone_OK := "_F209210ZS01Input".EStopSum,
                               I_AlarmA := "_209210ZM01".ZMS012AlarmA,
                               I_AlarmB := "_209210ZM01".ZMS012AlarmB,
                               I_AlarmC := "_209210ZM01".ZMS012AlarmC,
                               I_Modes := "_209210ZMS012Modes".Modes,
                               O_LED_Auto => "209210AS11PX1",
                               O_LED_Man => "209210AS11PX2",
                               O_LED_Fault => "209210AS11PX3",
                               O_LED_EStop => "209210AS11PX4");
   END_IF;
   IF "TRUE" THEN
       "LGBHWPanelLedIndication"(I_NumberHMI := 2,
                               I_ActiveHMI := "_209210ZMS013Modes".ActiveHMI,
                               I_EStopAS_OK := "_F209210ZS01Input"."210AS11F9SH1",
                               I_EStopZone_OK := "_F209210ZS01Input".EStopSum,
                               I_AlarmA := "_209210ZM01".ZMS013AlarmA,
                               I_AlarmB := "_209210ZM01".ZMS013AlarmB,
                               I_AlarmC := "_209210ZM01".ZMS013AlarmC,
                               I_Modes := "_209210ZMS013Modes".Modes,
                               O_LED_Auto => "209210AS11PX21",
                               O_LED_Man => "209210AS11PX22",
                               O_LED_Fault => "209210AS11PX23",
                               O_LED_EStop => "209210AS11PX24");
   END_IF;
END_REGION

REGION Network 33: **** 4.6 - Machine Status - Indication **** Stack Light 209210AS10
   IF "TRUE" THEN
       "_209210AS10StackLight"(I_ResetSafetyActive := "_209210ZS01Safety".ResetSafetyActive,   // "LGBStackLight"
                               IO_ModesZM1 := "_209210ZMS011Modes".Modes,
                               IO_ModesZM2 := "_209210ZMS012Modes".Modes,
                               IO_ModesZM3 := "_209210ZMS012Modes".Modes,
                               IO_ModesZM4 := "_209210ZMS012Modes".Modes,
                               IO_ModesZM5 := "_209210ZMS012Modes".Modes,
                               IO_ModesZM6 := "_209210ZMS012Modes".Modes,
                               IO_ModesZM7 := "_209210ZMS012Modes".Modes,
                               IO_ModesZM8 := "_209210ZMS012Modes".Modes,
                               IO_ModesZM9 := "_209210ZMS012Modes".Modes,
                               IO_ModesZM10 := "_209210ZMS012Modes".Modes,
                               IO_ModesZM11 := "_209210ZMS012Modes".Modes,
                               IO_ModesZM12 := "_209210ZMS012Modes".Modes,
                               IO_ModesZM13 := "_209210ZMS012Modes".Modes,
                               IO_ModesZM14 := "_209210ZMS012Modes".Modes,
                               IO_ModesZM15 := "_209210ZMS012Modes".Modes,
                               IO_ModesZM16 := "_209210ZMS012Modes".Modes,
                               O_AutoInd => "209210AS10P1PX1",
                               O_AlarmInd => "209210AS10P1PX2",
                               O_Buzzer => "209210AS10P1PA1");
   END_IF;
END_REGION

REGION Network 34: **** 4.6 - Machine Status - Indication **** Stack Light 209210AS11
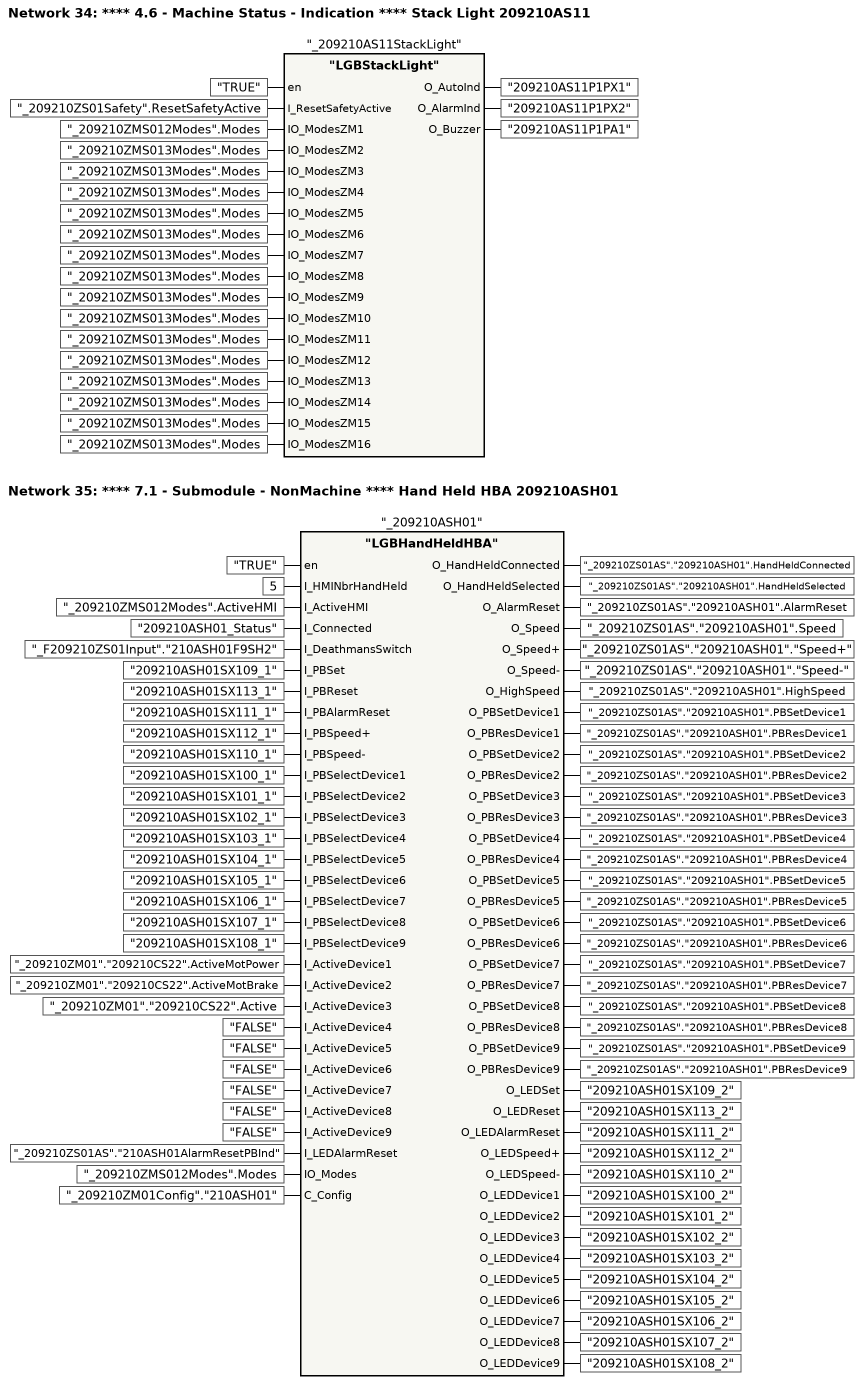
   IF "TRUE" THEN
       "_209210AS11StackLight"(I_ResetSafetyActive := "_209210ZS01Safety".ResetSafetyActive,   // "LGBStackLight"
                               IO_ModesZM1 := "_209210ZMS012Modes".Modes,
                               IO_ModesZM2 := "_209210ZMS013Modes".Modes,
                               IO_ModesZM3 := "_209210ZMS013Modes".Modes,
                               IO_ModesZM4 := "_209210ZMS013Modes".Modes,
                               IO_ModesZM5 := "_209210ZMS013Modes".Modes,
                               IO_ModesZM6 := "_209210ZMS013Modes".Modes,
                               IO_ModesZM7 := "_209210ZMS013Modes".Modes,
                               IO_ModesZM8 := "_209210ZMS013Modes".Modes,
                               IO_ModesZM9 := "_209210ZMS013Modes".Modes,
                               IO_ModesZM10 := "_209210ZMS013Modes".Modes,
                               IO_ModesZM11 := "_209210ZMS013Modes".Modes,
                               IO_ModesZM12 := "_209210ZMS013Modes".Modes,
                               IO_ModesZM13 := "_209210ZMS013Modes".Modes,
                               IO_ModesZM14 := "_209210ZMS013Modes".Modes,
                               IO_ModesZM15 := "_209210ZMS013Modes".Modes,
                               IO_ModesZM16 := "_209210ZMS013Modes".Modes,
                               O_AutoInd => "209210AS11P1PX1",
                               O_AlarmInd => "209210AS11P1PX2",
                               O_Buzzer => "209210AS11P1PA1");
   END_IF;
END_REGION

REGION Network 35: **** 7.1 - Submodule - NonMachine **** Hand Held HBA 209210ASH01
   IF "TRUE" THEN
       "_209210ASH01"(I_HMINbrHandHeld := 5,   // "LGBHandHeldHBA"
                      I_ActiveHMI := "_209210ZMS012Modes".ActiveHMI,
                      I_Connected := "209210ASH01_Status",
                      I_DeathmansSwitch := "_F209210ZS01Input"."210ASH01F9SH2",
                      I_PBSet := "209210ASH01SX109_1",
                      I_PBReset := "209210ASH01SX113_1",
                      I_PBAlarmReset := "209210ASH01SX111_1",
                      "I_PBSpeed+" := "209210ASH01SX112_1",
                      "I_PBSpeed-" := "209210ASH01SX110_1",
                      I_PBSelectDevice1 := "209210ASH01SX100_1",
                      I_PBSelectDevice2 := "209210ASH01SX101_1",
                      I_PBSelectDevice3 := "209210ASH01SX102_1",
                      I_PBSelectDevice4 := "209210ASH01SX103_1",
                      I_PBSelectDevice5 := "209210ASH01SX104_1",
                      I_PBSelectDevice6 := "209210ASH01SX105_1",
                      I_PBSelectDevice7 := "209210ASH01SX106_1",
                      I_PBSelectDevice8 := "209210ASH01SX107_1",
                      I_PBSelectDevice9 := "209210ASH01SX108_1",
                      I_ActiveDevice1 := "_209210ZM01"."209210CS22".ActiveMotPower,
                      I_ActiveDevice2 := "_209210ZM01"."209210CS22".ActiveMotBrake,
                      I_ActiveDevice3 := "_209210ZM01"."209210CS22".Active,
                      I_ActiveDevice4 := "FALSE",
                      I_ActiveDevice5 := "FALSE",
                      I_ActiveDevice6 := "FALSE",
                      I_ActiveDevice7 := "FALSE",
                      I_ActiveDevice8 := "FALSE",
                      I_ActiveDevice9 := "FALSE",
                      I_LEDAlarmReset := "_209210ZS01AS"."210ASH01AlarmResetPBInd",
                      IO_Modes := "_209210ZMS012Modes".Modes,
                      C_Config := "_209210ZM01Config"."210ASH01",
                      O_HandHeldConnected => "_209210ZS01AS"."209210ASH01".HandHeldConnected,
                      O_HandHeldSelected => "_209210ZS01AS"."209210ASH01".HandHeldSelected,
                      O_AlarmReset => "_209210ZS01AS"."209210ASH01".AlarmReset,
                      O_Speed => "_209210ZS01AS"."209210ASH01".Speed,
                      "O_Speed+" => "_209210ZS01AS"."209210ASH01"."Speed+",
                      "O_Speed-" => "_209210ZS01AS"."209210ASH01"."Speed-",
                      O_HighSpeed => "_209210ZS01AS"."209210ASH01".HighSpeed,
                      O_PBSetDevice1 => "_209210ZS01AS"."209210ASH01".PBSetDevice1,
                      O_PBResDevice1 => "_209210ZS01AS"."209210ASH01".PBResDevice1,
                      O_PBSetDevice2 => "_209210ZS01AS"."209210ASH01".PBSetDevice2,
                      O_PBResDevice2 => "_209210ZS01AS"."209210ASH01".PBResDevice2,
                      O_PBSetDevice3 => "_209210ZS01AS"."209210ASH01".PBSetDevice3,
                      O_PBResDevice3 => "_209210ZS01AS"."209210ASH01".PBResDevice3,
                      O_PBSetDevice4 => "_209210ZS01AS"."209210ASH01".PBSetDevice4,
                      O_PBResDevice4 => "_209210ZS01AS"."209210ASH01".PBResDevice4,
                      O_PBSetDevice5 => "_209210ZS01AS"."209210ASH01".PBSetDevice5,
                      O_PBResDevice5 => "_209210ZS01AS"."209210ASH01".PBResDevice5,
                      O_PBSetDevice6 => "_209210ZS01AS"."209210ASH01".PBSetDevice6,
                      O_PBResDevice6 => "_209210ZS01AS"."209210ASH01".PBResDevice6,
                      O_PBSetDevice7 => "_209210ZS01AS"."209210ASH01".PBSetDevice7,
                      O_PBResDevice7 => "_209210ZS01AS"."209210ASH01".PBResDevice7,
                      O_PBSetDevice8 => "_209210ZS01AS"."209210ASH01".PBSetDevice8,
                      O_PBResDevice8 => "_209210ZS01AS"."209210ASH01".PBResDevice8,
                      O_PBSetDevice9 => "_209210ZS01AS"."209210ASH01".PBSetDevice9,
                      O_PBResDevice9 => "_209210ZS01AS"."209210ASH01".PBResDevice9,
                      O_LEDSet => "209210ASH01SX109_2",
                      O_LEDReset => "209210ASH01SX113_2",
                      O_LEDAlarmReset => "209210ASH01SX111_2",
                      "O_LEDSpeed+" => "209210ASH01SX112_2",
                      "O_LEDSpeed-" => "209210ASH01SX110_2",
                      O_LEDDevice1 => "209210ASH01SX100_2",
                      O_LEDDevice2 => "209210ASH01SX101_2",
                      O_LEDDevice3 => "209210ASH01SX102_2",
                      O_LEDDevice4 => "209210ASH01SX103_2",
                      O_LEDDevice5 => "209210ASH01SX104_2",
                      O_LEDDevice6 => "209210ASH01SX105_2",
                      O_LEDDevice7 => "209210ASH01SX106_2",
                      O_LEDDevice8 => "209210ASH01SX107_2",
                      O_LEDDevice9 => "209210ASH01SX108_2");
   END_IF;
END_REGION

REGION Network 36: **** 8 - Outputs **** Led Indication 209210AS10 - Equipment
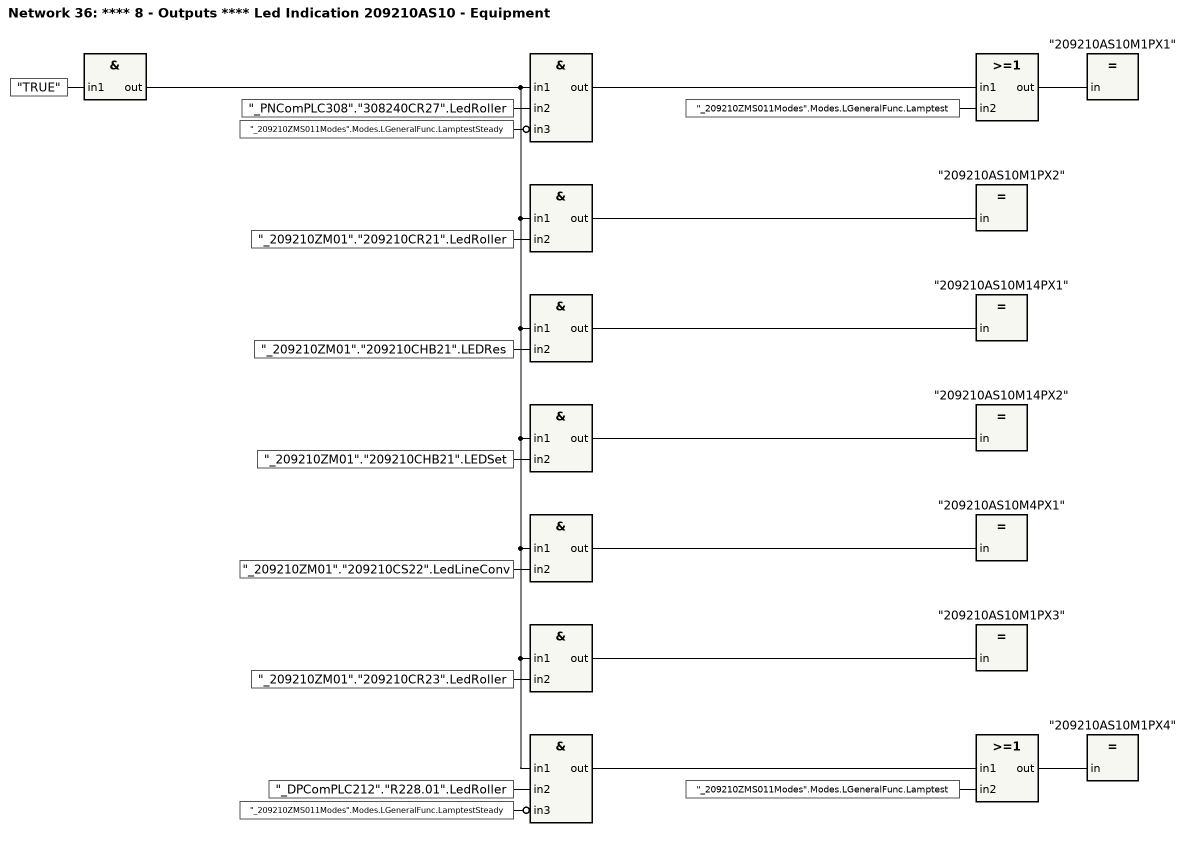
   "209210AS10M1PX1" := ("TRUE" AND "_PNComPLC308"."308240CR27".LedRoller AND NOT "_209210ZMS011Modes".Modes.LGeneralFunc.LamptestSteady) OR "_209210ZMS011Modes".Modes.LGeneralFunc.Lamptest;
   "209210AS10M1PX2" := "TRUE" AND "_209210ZM01"."209210CR21".LedRoller;
   "209210AS10M14PX1" := "TRUE" AND "_209210ZM01"."209210CHB21".LEDRes;
   "209210AS10M14PX2" := "TRUE" AND "_209210ZM01"."209210CHB21".LEDSet;
   "209210AS10M4PX1" := "TRUE" AND "_209210ZM01"."209210CS22".LedLineConv;
   "209210AS10M1PX3" := "TRUE" AND "_209210ZM01"."209210CR23".LedRoller;
   "209210AS10M1PX4" := ("TRUE" AND "_DPComPLC212"."R228.01".LedRoller AND NOT "_209210ZMS011Modes".Modes.LGeneralFunc.LamptestSteady) OR "_209210ZMS011Modes".Modes.LGeneralFunc.Lamptest;
END_REGION

REGION Network 37: **** 8 - Outputs **** Led Indication 209210AS11 - Equipment
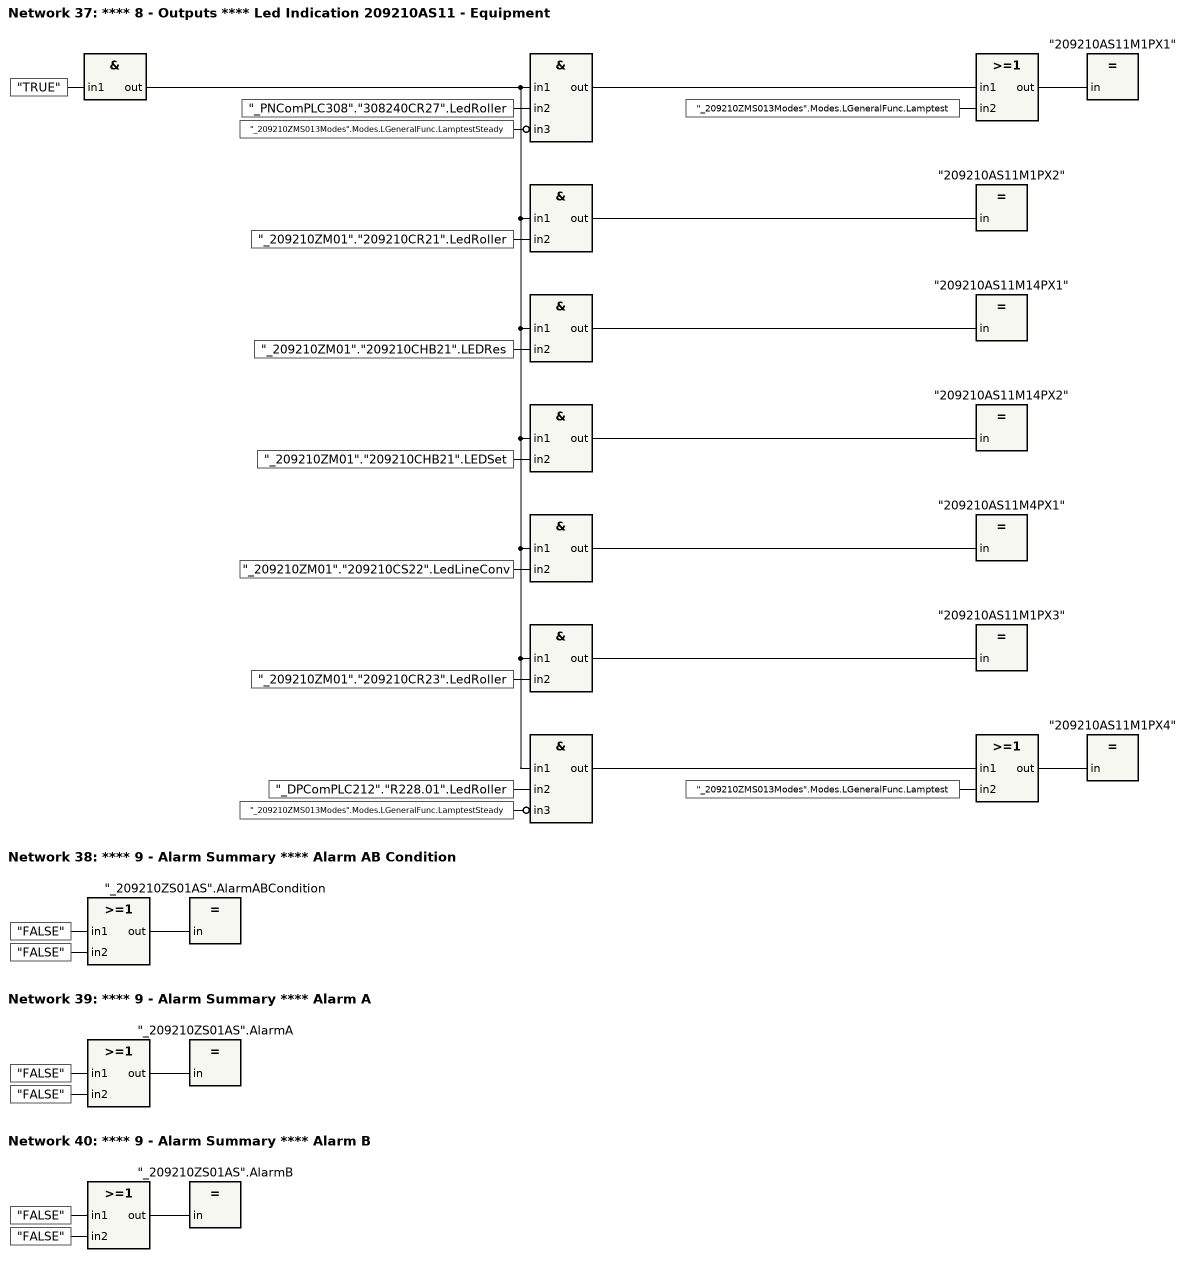
   "209210AS11M1PX1" := ("TRUE" AND "_PNComPLC308"."308240CR27".LedRoller AND NOT "_209210ZMS013Modes".Modes.LGeneralFunc.LamptestSteady) OR "_209210ZMS013Modes".Modes.LGeneralFunc.Lamptest;
   "209210AS11M1PX2" := "TRUE" AND "_209210ZM01"."209210CR21".LedRoller;
   "209210AS11M14PX1" := "TRUE" AND "_209210ZM01"."209210CHB21".LEDRes;
   "209210AS11M14PX2" := "TRUE" AND "_209210ZM01"."209210CHB21".LEDSet;
   "209210AS11M4PX1" := "TRUE" AND "_209210ZM01"."209210CS22".LedLineConv;
   "209210AS11M1PX3" := "TRUE" AND "_209210ZM01"."209210CR23".LedRoller;
   "209210AS11M1PX4" := ("TRUE" AND "_DPComPLC212"."R228.01".LedRoller AND NOT "_209210ZMS013Modes".Modes.LGeneralFunc.LamptestSteady) OR "_209210ZMS013Modes".Modes.LGeneralFunc.Lamptest;
END_REGION

REGION Network 38: **** 9 - Alarm Summary **** Alarm AB Condition
   // Alarm AB condition
   "_209210ZS01AS".AlarmABCondition := "FALSE" OR "FALSE";
END_REGION

REGION Network 39: **** 9 - Alarm Summary **** Alarm A
   // Summary of alarms A
   "_209210ZS01AS".AlarmA := "FALSE" OR "FALSE";
END_REGION

REGION Network 40: **** 9 - Alarm Summary **** Alarm B
   // Summary of alarms B
   "_209210ZS01AS".AlarmB := "FALSE" OR "FALSE";
END_REGION

REGION Network 41: **** 9 - Alarm Summary **** Alarm C
   // Summary of alarms C
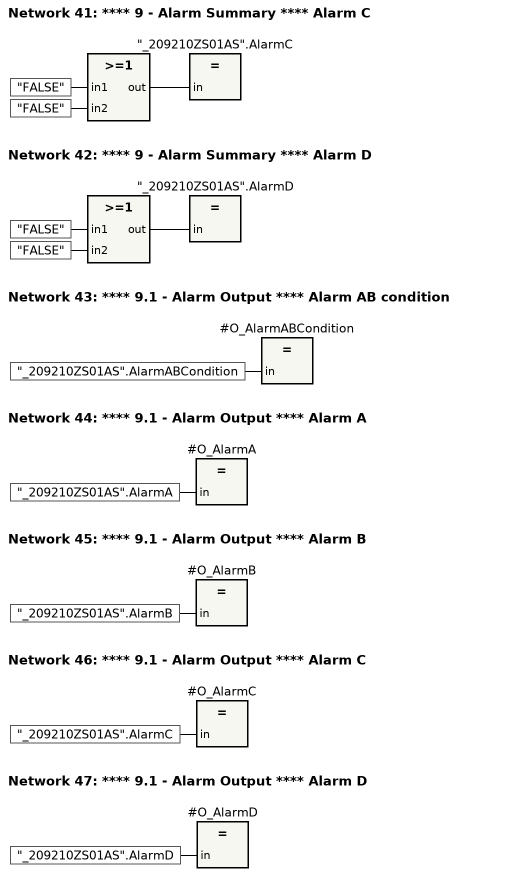
   "_209210ZS01AS".AlarmC := "FALSE" OR "FALSE";
END_REGION

REGION Network 42: **** 9 - Alarm Summary **** Alarm D
   // Summary of alarms D
   "_209210ZS01AS".AlarmD := "FALSE" OR "FALSE";
END_REGION

REGION Network 43: **** 9.1 - Alarm Output **** Alarm AB condition
   // Alarm AB condition
   #O_AlarmABCondition := "_209210ZS01AS".AlarmABCondition;
END_REGION

REGION Network 44: **** 9.1 - Alarm Output **** Alarm A
   // Output Alarm A
   #O_AlarmA := "_209210ZS01AS".AlarmA;
END_REGION

REGION Network 45: **** 9.1 - Alarm Output **** Alarm B
   // Output Alarm B
   #O_AlarmB := "_209210ZS01AS".AlarmB;
END_REGION

REGION Network 46: **** 9.1 - Alarm Output **** Alarm C
   // Output Alarm A
   #O_AlarmC := "_209210ZS01AS".AlarmC;
END_REGION

REGION Network 47: **** 9.1 - Alarm Output **** Alarm D
   // Output Alarm D
   #O_AlarmD := "_209210ZS01AS".AlarmD;
END_REGION

REGION Network 48: **** 9.2 - Alarm DWord**** Alarm To DWord
   // Alarm Word
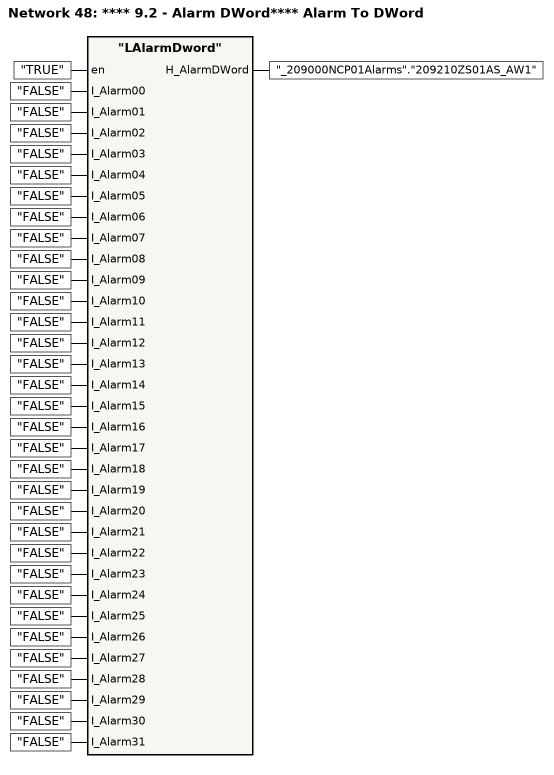
   IF "TRUE" THEN
       "LAlarmDword"(I_Alarm00 := "FALSE",
                     I_Alarm01 := "FALSE",
                     I_Alarm02 := "FALSE",
                     I_Alarm03 := "FALSE",
                     I_Alarm04 := "FALSE",
                     I_Alarm05 := "FALSE",
                     I_Alarm06 := "FALSE",
                     I_Alarm07 := "FALSE",
                     I_Alarm08 := "FALSE",
                     I_Alarm09 := "FALSE",
                     I_Alarm10 := "FALSE",
                     I_Alarm11 := "FALSE",
                     I_Alarm12 := "FALSE",
                     I_Alarm13 := "FALSE",
                     I_Alarm14 := "FALSE",
                     I_Alarm15 := "FALSE",
                     I_Alarm16 := "FALSE",
                     I_Alarm17 := "FALSE",
                     I_Alarm18 := "FALSE",
                     I_Alarm19 := "FALSE",
                     I_Alarm20 := "FALSE",
                     I_Alarm21 := "FALSE",
                     I_Alarm22 := "FALSE",
                     I_Alarm23 := "FALSE",
                     I_Alarm24 := "FALSE",
                     I_Alarm25 := "FALSE",
                     I_Alarm26 := "FALSE",
                     I_Alarm27 := "FALSE",
                     I_Alarm28 := "FALSE",
                     I_Alarm29 := "FALSE",
                     I_Alarm30 := "FALSE",
                     I_Alarm31 := "FALSE",
                     H_AlarmDWord => "_209000NCP01Alarms"."209210ZS01AS_AW1");
   END_IF;
END_REGION
END_FUNCTION
